// TIA Portal V18 export
TYPE "RCS_SysCycleTime_V1"
   STRUCT
      No : Array[0..21] of Real;   // [0]LastTime,[21]AverageTime
   END_STRUCT;
END_TYPE
